TYPE T_Ctrl_SIf_SLB_Cfg :
STRUCT
END_STRUCT
END_TYPE

(* stored: Version 1.1.0.1, ProductVersion 3.1.0.19
   DUT T_Ctrl_SIf_SLB_Cfg: Id {c260bc19-ea1d-4085-956a-edbec0686d65} *)
